{attribute 'qualified_only'}
VAR_GLOBAL
	eMode : E_Control_Mode := E_Control_Mode.OFF;
	eStatus : E_Status := E_Status.NOTREADY;
	fbTon : TON := ();
	bStartTimer : BOOL := FALSE;
	bTimerDone : BOOL;
END_VAR

(* stored: Version 1.1.0.1, ProductVersion 3.1.4024.12
   GVL G_ControlBox: Id {58d0ea5b-1b17-4931-b151-b15e0c6b313c} *)
